ABB RobotStudio station: RealController_Simulation.rsstnx

Station RealController_Simulation (saved by RobotStudio 22.2.10013.1)
Controller CRB15000_5_95
  mechanical unit ROB_1: CRB15000_5_95__02, 6 joints, base frame (0, 0, 0) mm
Layout (positions relative to the parent item):
  - CRB15000_5_95__02 [mechanism, from Robots\CRB15000_5_95__02.rslib] at (0, 0, 0) mm; joint values [0, 0, 0, 0, 0.5236, 0] (rad or m)
  - gripper_rg6 [part] at (597.47, 0, 837.78) mm, rotated rx 180 ry 60 rz 180 deg, size 75.5 x 155 x 263.6 mm
Attachment: gripper_rg6 is attached to CRB15000_5_95__02 / Link6
